// TIA Portal V17 export
// export: Created 2026-04-13T11:12:44.8812846Z, ExportSetting WithDefaults, DisplayName Totally Integrated Automation Portal, DisplayVersion V17 Update 4, DisplayName TIA Portal Openness, DisplayVersion V17 Update 4, DisplayName TIA Portal Version Control Interface, DisplayVersion V17, DisplayName SINAMICS Startdrive Advanced, DisplayVersion V17, DisplayName SINAMICS Startdrive G130, G150, S120, S150, SINAMICS MV, S210, DisplayVersion V17, DisplayName SINAMICS Startdrive G110M, G120, G120C, G120D, G120P, G115D, DisplayVersion V17, DisplayName STEP 7 Professional, DisplayVersion V17 Update 4, DisplayName STEP 7 Safety, DisplayVersion V17, DisplayName WinCC Professional, DisplayVersion V17 Update 4
FUNCTION_BLOCK "Modbus_Comm_Load"   // FB640, SCL
TITLE = Modbus port configuration
AUTHOR : SIMATIC
FAMILY : MODBUS
NAME : MBCOMLOA
VERSION : 5.0
// stored: IsIECCheckEnabled true, SetENOAutomatically false, UDAEnableTagReadback false
   VAR_INPUT
      REQ : Bool;   // Startet die Konfiguration für Modbus RTU Kommunikation / Activates the configuration for Modbus RTU communication
      PORT : PORT := 0;   // Kommunikationsport, Hardwarekennung / Communication port, Hardware Identifier
      BAUD : UDInt := 9600;   // Datenübertragungsrate / Transmission rate
      PARITY : UInt := 0;   // Parität / Parity
      FLOW_CTRL : UInt := 0;   // Flusskontrolle / Enables or disables flow control
      RTS_ON_DLY : UInt := 0;   // Wartezeit nach Aktivierung von RTS, vor Übertragung von Tx-Daten (ms) / Time to wait after activating RTS before transmission will be initiated
      RTS_OFF_DLY : UInt := 0;   // Wartezeit nach Übertragung von Tx-Daten, bevor RTS deaktiviert wird (ms) / Time to wait before de-activating RTS once transmission has been completed
      RESP_TO : UInt := 1000;   // Zeitdauer, die der Master auf ein Antworttelegramm wartet / Time period that the master waits for a response
   END_VAR
   VAR_OUTPUT
      DONE : Bool;   // Anweisung beendet ohne Fehler / Instruction finished without error
      ERROR : Bool;   // Anweisung beendet mit Fehler / Instruction finished with error
      STATUS : Word := W#16#7000;   // Detailllierte Fehlerinformation / Detailed error information
   END_VAR
   VAR_IN_OUT
      MB_DB : P2P_MB_BASE;   // Zeiger auf den Parameter MB_DB des Modbus_Master oder Modbus_Slave Instanz-DBs / Reference to the parameter MB_DB of Modbus_Master or Modbus_Slave instance DB
   END_VAR
   VAR
      ICHAR_GAP : Word;   // Anzahl der Bitzeiten zwischen den Zeichen / Inter-character gap
      RETRIES : Word;   // Anzahl Wiederholversuche bei Timeout / Number of retries in case of a timeout
      MODE : USInt := 16#00;   // Duplex-Betriebsart / Duplex operation mode
      LINE_PRE : USInt := 16#00;   // Vorbelegung der Empfangsleitung / Presetting of the receive line
      BRK_DET : USInt := 16#00;   // RS232 Break-Erkennung / RS232 BREAK Handling
      EN_DIAG_ALARM : Bool;   // Generierung von Diagnosemeldungen aktivieren / Enable diagnostic alarm generation
      STOP_BITS : USInt := 1;   // Number of STOP bits; 1=1 Stop bit; 2=2 Stop bits
      EN_SUPPLY_VOLT : Bool;   // Diagnose für fehlende Versorgungsspannung L+ einschalten / Enable supply voltage diagnostic
      b_e_REQ : Bool;   // Flankenbit für REQ / Edge flag for REQ
      y_state : SInt := 16#00;   // Status der Anweisung / State of instruction
      Send_Config { S7_SetPoint := 'True'} : Send_Config;   // Lokale Instanz der Anweisung Send_Config / Local instance of the instruction Send_Config
      Receive_Config { S7_SetPoint := 'True'} : Receive_Config;   // Lokale Instanz der Anweisung Receive_Config / Local instance of the instruction Receive_Config
      Receive_Conditions { S7_SetPoint := 'True'} : Receive_Conditions;   // Parameter für Receive_Config / Parameter for Receive_Config
      WRREC { S7_SetPoint := 'True'} : WRREC;   // Lokale Instanz der Anweisung WRREC / Local instance of the instruction WRREC
      RDREC { S7_SetPoint := 'True'} : RDREC;   // Lokale Instanz der Anweisung RDREC / Local instance of the instruction RDREC
      port_w_record { ExternalVisible := 'False'; S7_SetPoint := 'True'} : P2P_MB_PortData;   // Nur für internen Gebrauch / For internal use only
      err_record { ExternalVisible := 'False'; S7_SetPoint := 'True'} : P2P_RdEstat;   // Nur für internen Gebrauch / For internal use only
      ftrs_w_record { ExternalVisible := 'False'; S7_SetPoint := 'True'} : P2P_FeaturesData;   // Nur für internen Gebrauch / For internal use only
   END_VAR
BEGIN
END_FUNCTION_BLOCK
